# EPICS substitutions: viocs/si_ps/si_psApp/Db/sda0.substitutions
file "db/individual.db" {
    pattern { family, pos, num }
        { "SDA0", "01M1", "" }
        { "SDA0", "01M2", "" }
        { "SDA0", "05M1", "" }
        { "SDA0", "05M2", "" }
        { "SDA0", "09M1", "" }
        { "SDA0", "09M2", "" }
        { "SDA0", "13M1", "" }
        { "SDA0", "13M2", "" }
        { "SDA0", "17M1", "" }
        { "SDA0", "17M2", "" }
}
